TYPE DUT_TASKSTATE :
(
	Unassigned := 0,
	Assigned := 1,
	WaitingForSkillReady := 2,
	InProgress := 3,
	Done := 4,
	Aborted := 5,
	Error := 6
);
END_TYPE

(* stored: Version 1.1.0.1, ProductVersion 3.1.0.25
   DUT DUT_TASKSTATE: Id {572afb3a-f785-4488-b2cc-5f28b0d38f3c} *)
